{attribute 'qualified_only'}
{attribute 'strict'}
{attribute 'to_string'}
TYPE FILE_CONTENT_HANDLING_MODE :
(
	BINARY := Tc2_System.FOPEN_MODEBINARY, // opens the file in binary mode
	TEXT := Tc2_System.FOPEN_MODETEXT // opens the file in text mode
) DWORD;
END_TYPE

(* stored: Version 1.1.0.1
   DUT FILE_CONTENT_HANDLING_MODE: Id {3da98897-3c82-4e81-a81f-23145bb75889} *)
